FUNCTION_BLOCK FB_ReadTime
VAR_INPUT
	bReset 					:BOOL;	
	bSignalIn				:BOOL;
END_VAR
VAR_OUTPUT
	//Delta time in ms from Digital sensor to camera TCP
	aDeltaTimeMS			:ARRAY[0..GVL_Constant.ITEM_ARRAY_SIZE] OF UDINT;
	//Digital input sensor
	aDigitalSensorTime		:ARRAY[0..ITEM_ARRAY_SIZE] OF STRING;
	//Camera TCP port
	aTCPPortCameraTime		:ARRAY[0..ITEM_ARRAY_SIZE] OF STRING;
END_VAR
VAR
END_VAR

//Call Functions
M_SaveSensorTime();
M_SaveCameraTCPTime();
M_CalculateDeltaTime();

METHOD PUBLIC M_CalculateDeltaTime
VAR
	iDeltaTime			:INT;
	iNDeltaTime			:INT;
	rDeltaTrig			:R_TRIG;
	SavedCameraTime		:T_FILETIME;
	SavedSensorTime		:T_FILETIME;
	
END_VAR
//Get saved time from camera and sensor method
SavedCameraTime:=M_SaveCameraTCPTime();
SavedSensorTime:=M_SaveSensorTime();

//Trigger of camera tcp read complete. Uses same as camera as this is the last one to receive
rDeltaTrig(CLK:=PRG_TCPIP.fbReadFromCameraTCP.bReadComplete);

IF rDeltaTrig.Q THEN
	
	//Calculate delta time
	aDeltaTimeMS[iDeltaTime] :=  (F_CXSubTimeStamp(nTimeStampHiDW_A:=SavedCameraTime.dwHighDateTime,
													   nTimeStampHiDW_B:=SavedSensorTime.dwHighDateTime,
													   nTimeStampLoDW_A:=SavedCameraTime.dwLowDateTime,
													   nTimeStampLoDW_B:=SavedSensorTime.dwLowDateTime)/1000);
	iDeltaTime := iDeltaTime +1;
END_IF

//Reset registry
IF bReset THEN
	FOR iNDeltaTime := 0 TO GVL_Constant.ITEM_ARRAY_SIZE DO 
		aDeltaTimeMS[iNDeltaTime] := 0;
	END_FOR
	iDeltaTime := 0;
END_IF
END_METHOD

METHOD PUBLIC M_SaveCameraTCPTime : T_FILETIME
VAR
	rTCPPortCamera		:R_TRIG;
	iTCPPortCamera		:INT;
	iNTCPCamera			:INT;
	fbGetCameraTime		:FB_SystemTime;
END_VAR
//Trigger of camera tcp read complete
rTCPPortCamera(CLK:=PRG_TCPIP.fbReadFromCameraTCP.bReadComplete);

IF rTCPPortCamera.Q THEN
	aTCPPortCameraTime[iTCPPortCamera] := fbGetCameraTime.M_GetSystemTimeToString();
	
	fbGetCameraTime.fbSystemTime(timeLoDW=>M_SaveCameraTCPTime.dwLowDateTime,
    							 timeHiDW=>M_SaveCameraTCPTime.dwHighDateTime);
	
	iTCPPortCamera := iTCPPortCamera +1;
END_IF

//Reset registry
IF bReset THEN
	FOR iNTCPCamera := 0 TO GVL_Constant.ITEM_ARRAY_SIZE DO 
		aTCPPortCameraTime[iNTCPCamera] := '';
	END_FOR
	iTCPPortCamera := 0;
END_IF
END_METHOD

METHOD PUBLIC M_SaveSensorTime : T_FILETIME
VAR
	rDigitalSensorIn		:R_TRIG;
	iDigitalSensor			:INT;
	iNDigitalSensor			:INT;
	fbGetSensorTime			:FB_SystemTime;
END_VAR
//Trigger of sensor input
rDigitalSensorIn(CLK:=bSignalIn);

IF rDigitalSensorIn.Q THEN
	aDigitalSensorTime[iDigitalSensor] := fbGetSensorTime.M_GetSystemTimeToString();
	
	fbGetSensorTime.fbSystemTime(timeLoDW=>M_SaveSensorTime.dwLowDateTime,
    							 timeHiDW=>M_SaveSensorTime.dwHighDateTime);
								 
	iDigitalSensor := iDigitalSensor +1;
END_IF

//Reset registry
IF bReset THEN
	FOR iNDigitalSensor := 0 TO GVL_Constant.ITEM_ARRAY_SIZE DO 
		aDigitalSensorTime[iNDigitalSensor] := '';
	END_FOR
	iDigitalSensor := 0;
END_IF
END_METHOD

END_FUNCTION_BLOCK

(* stored: Version 1.1.0.1, ProductVersion 3.1.4024.12
   POU FB_ReadTime: Id {5faed61f-a29b-4c44-ac5a-b7ed64021721}, SpecialFunc None
   Method M_CalculateDeltaTime: Id {a5129a3c-0d36-4a82-bf14-e117a70e330a}
   Method M_SaveCameraTCPTime: Id {9f3cdf40-e788-4c90-aed5-163aedc53860}
   Method M_SaveSensorTime: Id {cd1a26d1-d744-4b0d-8d44-8a38ddfb04e9} *)
